Staubli VAL3: homing.pgx

public program homing(num x_nAxisNum, bool& x_bRes)
  local bool l_bError
  local num l_nEtape
  local string l_sMsg
  local num l_nTps
  local bool l_bVerrou
  local bool l_bOK
  local num l_nDuration
  local string l_sYN[2]
  local num l_nDrvPos
begin
  //指定外部轴零点
  //  if !isPowered()
  //    popUpMsg("请先上电")
  //    return
  //  endIf
  //  x_bRes=false
  //  doStartHoming[x_nAxisNum]=false
  //  delay(0.1)
  //  aioSet(aoWorkMode[x_nAxisNum],6)
  //  doStartHoming[x_nAxisNum]=true
  //  l_sYN[0]="是"
  //  l_sYN[1]="否"
  //  if watch(diHomingReached[x_nAxisNum]==true,2)
  //    x_bRes=true
  //    popUpMsg("设置成功")
  //  endIf

  //
  x_bRes=false
  if !isPowered()
    popUpMsg("请先给机器人上电")
    return
  endIf
  doStartHoming[x_nAxisNum]=false
  aioSet(aoWorkMode[x_nAxisNum],cst:nHOMINGMODE)
  delay(0.1)
  doStartHoming[x_nAxisNum]=true
  wait(diHomingReached[x_nAxisNum]==false)
  wait(diHomingReached[x_nAxisNum]==true)
  disablePower()
  delay(0.1)
  aioSet(aoWorkMode[x_nAxisNum],cst:nINTERPMODE)
  x_bRes=true
end
